// TIA Portal V18 export
TYPE "ModeGenStruct"
// stored: IsFailsafeCompliant false
   STRUCT
      Out { S7_SetPoint := 'True'} : "ModeOutStruct";
   END_STRUCT;
END_TYPE
